(* IEC 61131-3 sources: robotics-sec-platform/vm-ot/openplc, 3 files *)

(* ---- demo_jog.st ---- *)
(* SIGNED_BY: lab-release@lab.local @ 2026-06-06T12:00:00Z *)
(* Demo jog routine for the lab robot arm (hardened version - passes all gates). *)

PROGRAM JOG_CONTROL
  VAR_INPUT
    jog_request   : BOOL;
    e_stop_active : BOOL;
    safety_ok     : BOOL;
  END_VAR
  VAR_OUTPUT
    jog_allowed : BOOL;
  END_VAR
  VAR
    i : UINT;
  END_VAR

  (* Motion is permitted only when the E-stop is clear AND the safety supervisor agrees. *)
  IF jog_request AND NOT e_stop_active AND SAFETY_OK THEN
      jog_allowed := TRUE;
      FOR i := 0 TO 50 DO                    (* bounded by a static literal *)
          jog_allowed := TRUE;
      END_FOR;
  ELSE
      jog_allowed := FALSE;
  END_IF;

END_PROGRAM

PROGRAM SAFETY_JOG_OUTPUT
  VAR_INPUT
    jog_allowed   : BOOL;
    e_stop_active : BOOL;
  END_VAR
  (* Safety-owned block: ONLY here may the %QX0.x safety output be driven. *)
  IF jog_allowed AND NOT e_stop_active AND SAFETY_OK THEN
      %QX0.0 := TRUE;
  ELSE
      %QX0.0 := FALSE;
  END_IF;
END_PROGRAM

(* ---- production.st ---- *)
(* SIGNED_BY: lab-release@lab.local @ 2026-05-19T22:00:00Z *)
(* ===================================================================== *)
(* PRODUCTION PLC ladder logic for the lab cell                          *)
(*                                                                       *)
(* IEC 61131-3 Structured Text (.st) loaded by OpenPLC v3 (iec2c).       *)
(* Modbus mapping (OpenPLC standard):                                    *)
(*   Discrete Inputs  %IX0.0..%IX1.7  -> Modbus addresses 0..15          *)
(*   Coils            %QX0.0..%QX1.7  -> Modbus addresses 0..15          *)
(*   Holding Regs     %MW0..%MW63     -> Modbus addresses 0..63          *)
(*                                                                       *)
(* What this program does:                                               *)
(*   - 6-step pick-and-place state machine driven by a 100 ms scan.      *)
(*   - Publishes step + cycle counter on holding registers (telemetry).  *)
(*   - Honours an E-stop (%IX0.2) AND a "request_safe_state" (%IX0.3)    *)
(*     coil that the Stage-3 Safety Supervisor will assert via SROS2.    *)
(*   - Counts E-stop trips for Stage-6 incident metrics.                 *)
(*                                                                       *)
(* Notes for the iec2c front-end:                                        *)
(*   * VAR blocks are split by category (located inputs, located outputs,*)
(*     located memory words, plain internals) because iec2c is picky     *)
(*     about mixing AT-located and plain declarations in one block.      *)
(*   * TON instances are always called with both IN and PT parameters    *)
(*     in one statement; partial calls confuse the parser.               *)
(* ===================================================================== *)

PROGRAM PRODUCTION_PROGRAM
  VAR
    cycle_start_btn AT %IX0.0 : BOOL;
    cycle_stop_btn AT %IX0.1 : BOOL;
  END_VAR

  VAR
    motor_arm_enable AT %QX0.0 : BOOL;
    gripper_close AT %QX0.1 : BOOL;
    conveyor_run AT %QX0.2 : BOOL;
    cycle_busy AT %QX0.3 : BOOL;
    cycle_complete AT %QX0.4 : BOOL;
    e_stop_active AT %QX0.5 : BOOL;
    request_safe_state AT %QX0.6 : BOOL;
    remote_start_btn AT %QX1.0 : BOOL;
    remote_stop_btn AT %QX1.1 : BOOL;
  END_VAR

  VAR
    cycle_step AT %MW0 : UINT;
    cycle_count AT %MW1 : UINT;
    estop_trip_count AT %MW2 : UINT;
    last_cycle_ms AT %MW3 : UINT;
    slow_mode_active AT %MW4 : UINT;
    safety_state AT %MW10 : UINT;
    last_fault_code AT %MW12 : UINT;
  END_VAR

  VAR
    step_timer           : TON;
    last_estop           : BOOL;
    step_run             : BOOL;
    step_pt              : TIME;
    safe_state_now       : BOOL;
    cycle_running        : BOOL;
  END_VAR

  (* ------------------------------------------------------------------ *)
  (* SAFETY-FIRST INTERLOCK                                              *)
  (* If E-stop or safe-state asserted: drop everything, hold step 0.     *)
  (* ------------------------------------------------------------------ *)
  safe_state_now := e_stop_active OR request_safe_state;

  IF safe_state_now THEN
    motor_arm_enable := FALSE;
    gripper_close    := FALSE;
    conveyor_run     := FALSE;
    cycle_busy       := FALSE;
    cycle_step       := 0;
    step_run         := FALSE;
    cycle_running    := FALSE;
    IF e_stop_active AND NOT last_estop THEN
      estop_trip_count := estop_trip_count + 1;
    END_IF;
  END_IF;
  last_estop := e_stop_active;

  (* ------------------------------------------------------------------ *)
  (* CYCLE STATE MACHINE                                                 *)
  (*   step 0: idle, wait for start                                      *)
  (*   step 1: convey part into cell  (1.0 s)                            *)
  (*   step 2: arm moves to pick      (1.5 s)                            *)
  (*   step 3: gripper close          (0.5 s)                            *)
  (*   step 4: arm moves to place     (1.5 s)                            *)
  (*   step 5: gripper open           (0.5 s)                            *)
  (*   step 6: complete pulse                                            *)
  (* ------------------------------------------------------------------ *)
  IF NOT safe_state_now THEN

    (* Per-step actions (outputs) and the PT for the per-step timer.    *)
    CASE cycle_step OF
      0:
        cycle_busy       := FALSE;
        cycle_complete   := FALSE;
        conveyor_run     := FALSE;
        gripper_close    := FALSE;
        motor_arm_enable := FALSE;
        step_pt := T#100ms;
      1:
        conveyor_run     := TRUE;
        motor_arm_enable := TRUE;
        IF slow_mode_active = 1 THEN
          step_pt := T#2000ms;
        ELSE
          step_pt := T#1000ms;
        END_IF;
      2:
        conveyor_run     := FALSE;
        motor_arm_enable := TRUE;
        IF slow_mode_active = 1 THEN
          step_pt := T#3000ms;
        ELSE
          step_pt := T#1500ms;
        END_IF;
      3:
        gripper_close    := TRUE;
        IF slow_mode_active = 1 THEN
          step_pt := T#1000ms;
        ELSE
          step_pt := T#500ms;
        END_IF;
      4:
        IF slow_mode_active = 1 THEN
          step_pt := T#3000ms;
        ELSE
          step_pt := T#1500ms;
        END_IF;
      5:
        gripper_close    := FALSE;
        IF slow_mode_active = 1 THEN
          step_pt := T#1000ms;
        ELSE
          step_pt := T#500ms;
        END_IF;
      6:
        cycle_complete   := TRUE;
        IF NOT cycle_running THEN
          cycle_busy     := FALSE;
        END_IF;
        motor_arm_enable := FALSE;
        step_pt := T#100ms;
    END_CASE;

    (* Timer tick. Always called once per scan with current step_pt.    *)
    step_timer(IN := step_run, PT := step_pt);

    IF cycle_step = 0 THEN
      step_run := FALSE;
      IF (cycle_start_btn OR remote_start_btn) AND NOT (cycle_stop_btn OR remote_stop_btn) THEN
        cycle_step    := 1;
        cycle_busy    := TRUE;
        step_run      := TRUE;
        cycle_running := TRUE;
      END_IF;
    ELSIF step_timer.Q THEN
      (* Re-arm the timer for the next step. *)
      step_run := FALSE;
      IF cycle_step = 6 THEN
        cycle_count    := cycle_count + 1;
        last_cycle_ms  := 6100; (* nominal full-cycle ms; precise meas in Stage 2 *)
        IF cycle_running AND NOT (cycle_stop_btn OR remote_stop_btn) THEN
          cycle_step  := 1;
          step_run    := TRUE;
        ELSE
          cycle_step  := 0;
          cycle_busy  := FALSE;
        END_IF;
      ELSE
        cycle_step := cycle_step + 1;
        step_run   := TRUE;
      END_IF;
    END_IF;

    (* Handle cycle abort / stop *)
    IF cycle_stop_btn OR remote_stop_btn THEN
      cycle_running := FALSE;
      IF cycle_step > 0 THEN
        cycle_step := 0;
        cycle_busy := FALSE;
        step_run   := FALSE;
      END_IF;
    END_IF;

    (* Reset momentary buttons *)
    remote_start_btn := FALSE;
    remote_stop_btn  := FALSE;

  END_IF;

END_PROGRAM

(* ===================================================================== *)
(* CONFIGURATION + TASK BINDING                                          *)
(* ===================================================================== *)
CONFIGURATION Config0
  RESOURCE Res0 ON PLC
    TASK MAIN_TASK(INTERVAL := T#100ms, PRIORITY := 0);
    PROGRAM main_inst WITH MAIN_TASK : PRODUCTION_PROGRAM;
  END_RESOURCE
END_CONFIGURATION

(* ---- safety_supervisor.st ---- *)
(* SIGNED_BY: lab-release@lab.local @ 2026-05-19T22:00:00Z *)
(*
 * Safety Supervisor — IEC 61131-3 Structured Text reference ladder.
 *
 * This file is the *normative specification* of the safety logic. The
 * lab actually executes the same logic in Python (see
 * vm-ot/sros2/safety_supervisor.py) so we can co-locate the SROS2
 * (DDS) authentication layer in one process. The Python implementation
 * mirrors this ST file rung-for-rung; any change here MUST be reflected
 * there. Use this file as the artifact you would deploy to a real
 * second OpenPLC (192.168.10.11:503) when porting to hardware.
 *
 * Inputs  (Modbus holding registers received from production PLC):
 *   %MW0  hb_counter      : monotonic heartbeat (1 Hz baseline, 5 Hz under load)
 *   %MW1  prod_state      : production PLC operating state (0=idle, 1=run, 2=fault)
 *   %MW2  remote_estop    : 1 if a (cryptographically authenticated) remote E-stop was issued
 *
 * Outputs (Modbus holding registers polled by the runtime to publish /safety/state):
 *   %MW10 safety_state    : 0=NORMAL, 1=DEGRADED, 2=EMERGENCY
 *   %MW11 ack_counter     : echoes hb_counter when last accepted
 *   %MW12 last_fault_code : reason for the most recent EMERGENCY transition
 *
 * Fault codes (last_fault_code):
 *   0  no fault
 *   1  heartbeat watchdog (no hb_counter increment within HB_TIMEOUT)
 *   2  production reported its own fault (prod_state == 2)
 *   3  authenticated remote E-stop request
 *   4  invalid hb_counter sequence (replay/regression)
 *)

PROGRAM SafetySupervisor

  VAR_INPUT
    hb_counter   : UINT;
    prod_state   : UINT;
    remote_estop : BOOL;
  END_VAR

  VAR_OUTPUT
    safety_state    : UINT := 0;     (* NORMAL *)
    ack_counter     : UINT := 0;
    last_fault_code : UINT := 0;
  END_VAR

  VAR
    last_hb         : UINT := 0;
    hb_watchdog     : TON;
    hb_changed      : BOOL := FALSE;
  END_VAR

  (* --- 1. Detect a fresh heartbeat (counter incremented since last scan). *)
  hb_changed := (hb_counter <> last_hb) AND (hb_counter > last_hb);

  (* --- 2. Replay/regression guard: counter must monotonically increase. *)
  IF (hb_counter < last_hb) AND (last_hb - hb_counter < 1000) THEN
      safety_state    := 2;          (* EMERGENCY *)
      last_fault_code := 4;
  END_IF;

  (* --- 3. Heartbeat watchdog. Reset on each fresh hb. *)
  hb_watchdog(IN := NOT hb_changed, PT := T#500ms);

  IF hb_watchdog.Q AND (safety_state <> 2) THEN
      safety_state    := 2;
      last_fault_code := 1;
  END_IF;

  (* --- 4. Production self-reported fault. *)
  IF prod_state = 2 THEN
      safety_state    := 2;
      last_fault_code := 2;
  END_IF;

  (* --- 5. Authenticated remote E-stop. *)
  IF remote_estop THEN
      safety_state    := 2;
      last_fault_code := 3;
  END_IF;

  (* --- 6. Once EMERGENCY is latched it must remain latched until the
   *       supervisor process is restarted. There is no "auto-clear"
   *       transition from EMERGENCY back to NORMAL inside this scan. *)

  (* --- 7. Health bookkeeping for diagnostics. *)
  IF hb_changed THEN
      ack_counter := hb_counter;
      last_hb     := hb_counter;
  END_IF;

END_PROGRAM

CONFIGURATION Config0

  RESOURCE Res0 ON PLC
    TASK SafetyTask(INTERVAL := T#50ms, PRIORITY := 0);
    PROGRAM SafetyInst WITH SafetyTask : SafetySupervisor;
  END_RESOURCE

END_CONFIGURATION
